Staubli VAL3: ONACTION.pgx

program OnAction()
  local num l_nX
  local num l_nY
begin
  //示教动作
  //示教动作执行

  wait(isPowered())
  for l_nX=0 to 11
    for l_nY=0 to 1
     Motion:nMoveidAction[l_nX,l_nY]=TxtFile:nAction[nTeachAction,l_nX,l_nY]

    endFor
  endFor


  call IO:Action(Motion:nMoveidAction,true,-1)
  call IO:Action(Motion:nMoveidAction,false,-1)


end
